FUNCTION_BLOCK CHECKPOINT_CAT (* Composite Function Block Type *)
  (* Standard: 61499-2 *)
  (* Version 0.0, 12/17/2022, Dmitrii, Flexbridge AB, template *)
  PACKAGE Main;
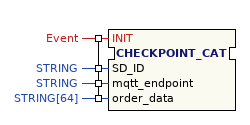
  EVENT_INPUT
    INIT WITH SD_ID, mqtt_endpoint, order_data;
  END_EVENT
  VAR_INPUT
    SD_ID : STRING;
    mqtt_endpoint : STRING;
    order_data : STRING[64]; (* Indication Data from Plug *)
  END_VAR
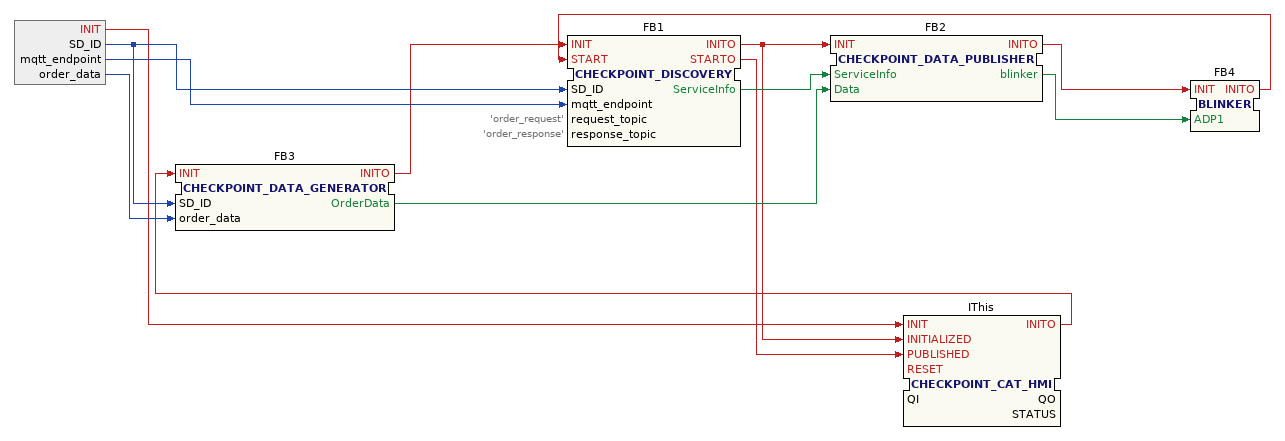
  (* Discovery & publish interface *)
  FBS
    FB1 : CHECKPOINT_DISCOVERY(request_topic := 'order_request', response_topic := 'order_response');
    FB2 : CHECKPOINT_DATA_PUBLISHER;
    FB3 : CHECKPOINT_DATA_GENERATOR;
    FB4 : BLINKER;
    IThis : CHECKPOINT_CAT_HMI;
  END_FBS
  EVENT_CONNECTIONS
    FB3.INITO TO FB1.INIT;
    FB1.INITO TO FB2.INIT;
    FB2.INITO TO FB4.INIT;
    FB4.INITO TO FB1.START;
    INIT TO IThis.INIT;
    FB1.INITO TO IThis.INITIALIZED;
    FB1.STARTO TO IThis.PUBLISHED;
    IThis.INITO TO FB3.INIT;
  END_CONNECTIONS
  DATA_CONNECTIONS
    SD_ID TO FB1.SD_ID;
    SD_ID TO FB3.SD_ID;
    mqtt_endpoint TO FB1.mqtt_endpoint;
    order_data TO FB3.order_data;
  END_CONNECTIONS
  ADAPTER_CONNECTIONS
    FB1.ServiceInfo TO FB2.ServiceInfo;
    FB3.OrderData TO FB2.Data;
    FB2.blinker TO FB4.ADP1;
  END_CONNECTIONS
END_FUNCTION_BLOCK
